TYPE T_Ctrl_SIf_COS_Cfg :
STRUCT
END_STRUCT
END_TYPE

(* stored: Version 1.1.0.1, ProductVersion 3.1.0.36
   DUT T_Ctrl_SIf_COS_Cfg: Id {0ec505fd-e7e4-42be-95e0-d1340e176b03} *)
